// TIA Portal V21 export
FUNCTION "PHT_Logic" : Void   // FC1206, LAD
{ S7_Optimized_Access := 'FALSE' }
// stored: AutoNumber false, SetENOAutomatically false
   VAR_TEMP   // added for the SCL form of the ladder/FBD networks
      _w1 : Bool;
      _w2 : Bool;
      _w3 : Bool;
      _w4 : Bool;
      _w5 : Bool;
      _w6 : Bool;
      _w7 : Bool;
   END_VAR
BEGIN

REGION Network 1: "PHT Cycle".Start
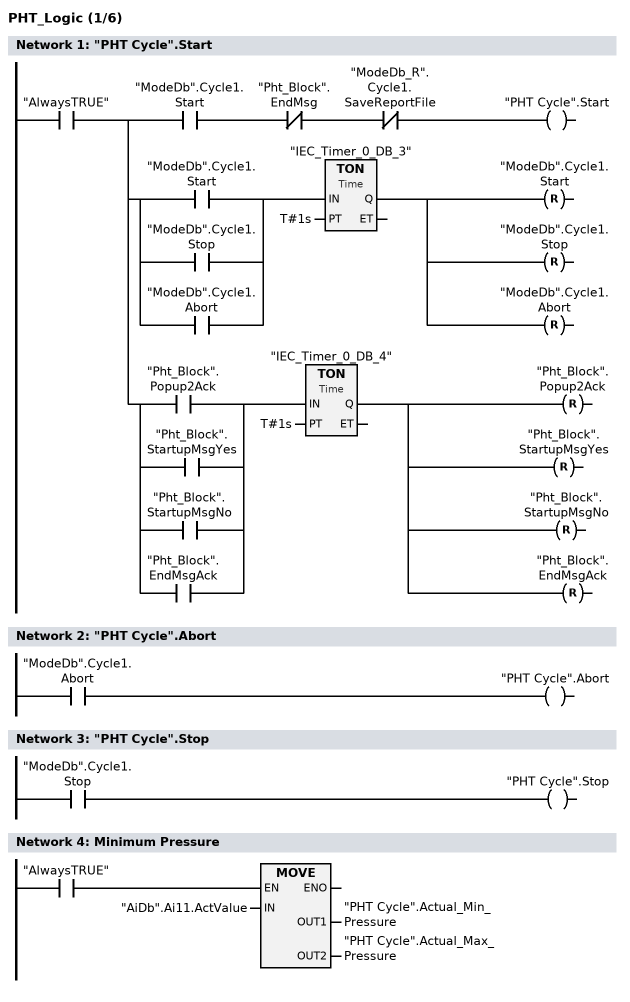
   RUNG wire#powerrail
      Contact( "AlwaysTRUE" )
      wire#w1
      Contact( "ModeDb".Cycle1.Start )
      I_Contact( "Pht_Block".EndMsg )
      I_Contact( "ModeDb_R".Cycle1.SaveReportFile )
      Coil( "PHT Cycle".Start )
   END_RUNG
   RUNG wire#w1
      Contact( "ModeDb".Cycle1.Start )
      wire#w2
      { S7_Templates := "time_type := Time" } "IEC_Timer_0_DB_3".TON(pt := T#1s, et =>)
      wire#w3
      R_Coil( "ModeDb".Cycle1.Start )
   END_RUNG
   RUNG wire#w1
      Contact( "ModeDb".Cycle1.Stop )
   END_RUNG wire#w2
   RUNG wire#w1
      Contact( "ModeDb".Cycle1.Abort )
   END_RUNG wire#w2
   RUNG wire#w3
      R_Coil( "ModeDb".Cycle1.Stop )
   END_RUNG
   RUNG wire#w3
      R_Coil( "ModeDb".Cycle1.Abort )
   END_RUNG
   RUNG wire#w1
      Contact( "Pht_Block".Popup2Ack )
      wire#w4
      { S7_Templates := "time_type := Time" } "IEC_Timer_0_DB_4".TON(pt := T#1s, et =>)
      wire#w5
      R_Coil( "Pht_Block".Popup2Ack )
   END_RUNG
   RUNG wire#w1
      Contact( "Pht_Block".StartupMsgYes )
   END_RUNG wire#w4
   RUNG wire#w1
      Contact( "Pht_Block".StartupMsgNo )
   END_RUNG wire#w4
   RUNG wire#w1
      Contact( "Pht_Block".EndMsgAck )
   END_RUNG wire#w4
   RUNG wire#w5
      R_Coil( "Pht_Block".StartupMsgYes )
   END_RUNG
   RUNG wire#w5
      R_Coil( "Pht_Block".StartupMsgNo )
   END_RUNG
   RUNG wire#w5
      R_Coil( "Pht_Block".EndMsgAck )
   END_RUNG
   // the same network as SCL:
   "PHT Cycle".Start := "AlwaysTRUE" AND "ModeDb".Cycle1.Start AND NOT "Pht_Block".EndMsg AND NOT "ModeDb_R".Cycle1.SaveReportFile;
   "IEC_Timer_0_DB_3".TON(IN := "AlwaysTRUE" AND ("ModeDb".Cycle1.Start OR "ModeDb".Cycle1.Stop OR "ModeDb".Cycle1.Abort),
                          PT := T#1s);
   IF "IEC_Timer_0_DB_3".Q THEN
       "ModeDb".Cycle1.Start := FALSE;
       "ModeDb".Cycle1.Stop := FALSE;
       "ModeDb".Cycle1.Abort := FALSE;
   END_IF;
   "IEC_Timer_0_DB_4".TON(IN := "AlwaysTRUE" AND ("Pht_Block".Popup2Ack OR "Pht_Block".StartupMsgYes OR "Pht_Block".StartupMsgNo OR "Pht_Block".EndMsgAck),
                          PT := T#1s);
   IF "IEC_Timer_0_DB_4".Q THEN
       "Pht_Block".Popup2Ack := FALSE;
       "Pht_Block".StartupMsgYes := FALSE;
       "Pht_Block".StartupMsgNo := FALSE;
       "Pht_Block".EndMsgAck := FALSE;
   END_IF;
END_REGION

REGION Network 2: "PHT Cycle".Abort
   RUNG wire#powerrail
      Contact( "ModeDb".Cycle1.Abort )
      Coil( "PHT Cycle".Abort )
   END_RUNG
   // the same network as SCL:
   "PHT Cycle".Abort := "ModeDb".Cycle1.Abort;
END_REGION

REGION Network 3: "PHT Cycle".Stop
   RUNG wire#powerrail
      Contact( "ModeDb".Cycle1.Stop )
      Coil( "PHT Cycle".Stop )
   END_RUNG
   // the same network as SCL:
   "PHT Cycle".Stop := "ModeDb".Cycle1.Stop;
END_REGION

REGION Network 4: Minimum Pressure
   RUNG wire#powerrail
      Contact( "AlwaysTRUE" )
      Move(in := "AiDb".Ai11.ActValue, out1 => "PHT Cycle".Actual_Min_Pressure, out2 => "PHT Cycle".Actual_Max_Pressure)
   END_RUNG
   // the same network as SCL:
   IF "AlwaysTRUE" THEN
       "PHT Cycle".Actual_Min_Pressure := "AiDb".Ai11.ActValue;
       "PHT Cycle".Actual_Max_Pressure := "AiDb".Ai11.ActValue;
   END_IF;
END_REGION

REGION Network 5: "PHT Cycle".fault
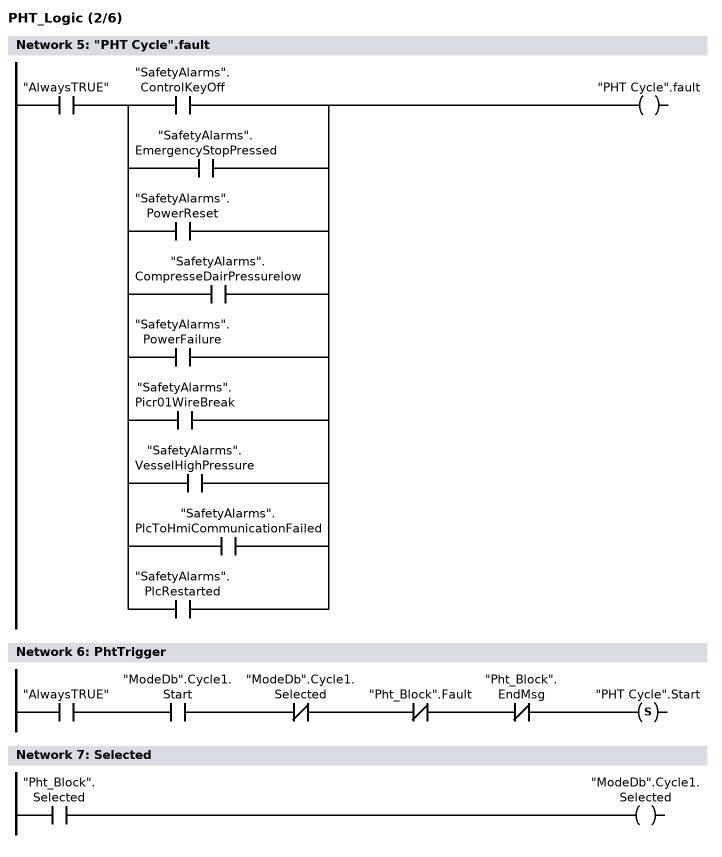
   RUNG wire#powerrail
      Contact( "AlwaysTRUE" )
      wire#w1
      Contact( "SafetyAlarms".ControlKeyOff )
      wire#w2
      Coil( "PHT Cycle".fault )
   END_RUNG
   RUNG wire#w1
      Contact( "SafetyAlarms".EmergencyStopPressed )
   END_RUNG wire#w2
   RUNG wire#w1
      Contact( "SafetyAlarms".PowerReset )
   END_RUNG wire#w2
   RUNG wire#w1
      Contact( "SafetyAlarms".CompresseDairPressurelow )
   END_RUNG wire#w2
   RUNG wire#w1
      Contact( "SafetyAlarms".PowerFailure )
   END_RUNG wire#w2
   RUNG wire#w1
      Contact( "SafetyAlarms".Picr01WireBreak )
   END_RUNG wire#w2
   RUNG wire#w1
      Contact( "SafetyAlarms".VesselHighPressure )
   END_RUNG wire#w2
   RUNG wire#w1
      Contact( "SafetyAlarms".PlcToHmiCommunicationFailed )
   END_RUNG wire#w2
   RUNG wire#w1
      Contact( "SafetyAlarms".PlcRestarted )
   END_RUNG wire#w2
   // the same network as SCL:
   "PHT Cycle".fault := "AlwaysTRUE" AND ("SafetyAlarms".ControlKeyOff OR "SafetyAlarms".EmergencyStopPressed OR "SafetyAlarms".PowerReset OR "SafetyAlarms".CompresseDairPressurelow OR "SafetyAlarms".PowerFailure OR "SafetyAlarms".Picr01WireBreak OR "SafetyAlarms".VesselHighPressure OR "SafetyAlarms".PlcToHmiCommunicationFailed OR "SafetyAlarms".PlcRestarted);
END_REGION

REGION Network 6: PhtTrigger
   RUNG wire#powerrail
      Contact( "AlwaysTRUE" )
      Contact( "ModeDb".Cycle1.Start )
      I_Contact( "ModeDb".Cycle1.Selected )
      I_Contact( "Pht_Block".Fault )
      I_Contact( "Pht_Block".EndMsg )
      S_Coil( "PHT Cycle".Start )
   END_RUNG
   // the same network as SCL:
   IF "AlwaysTRUE" AND "ModeDb".Cycle1.Start AND NOT "ModeDb".Cycle1.Selected AND NOT "Pht_Block".Fault AND NOT "Pht_Block".EndMsg THEN
       "PHT Cycle".Start := TRUE;
   END_IF;
END_REGION

REGION Network 7: Selected
   RUNG wire#powerrail
      Contact( "Pht_Block".Selected )
      Coil( "ModeDb".Cycle1.Selected )
   END_RUNG
   // the same network as SCL:
   "ModeDb".Cycle1.Selected := "Pht_Block".Selected;
END_REGION

REGION Network 8: PHT Block
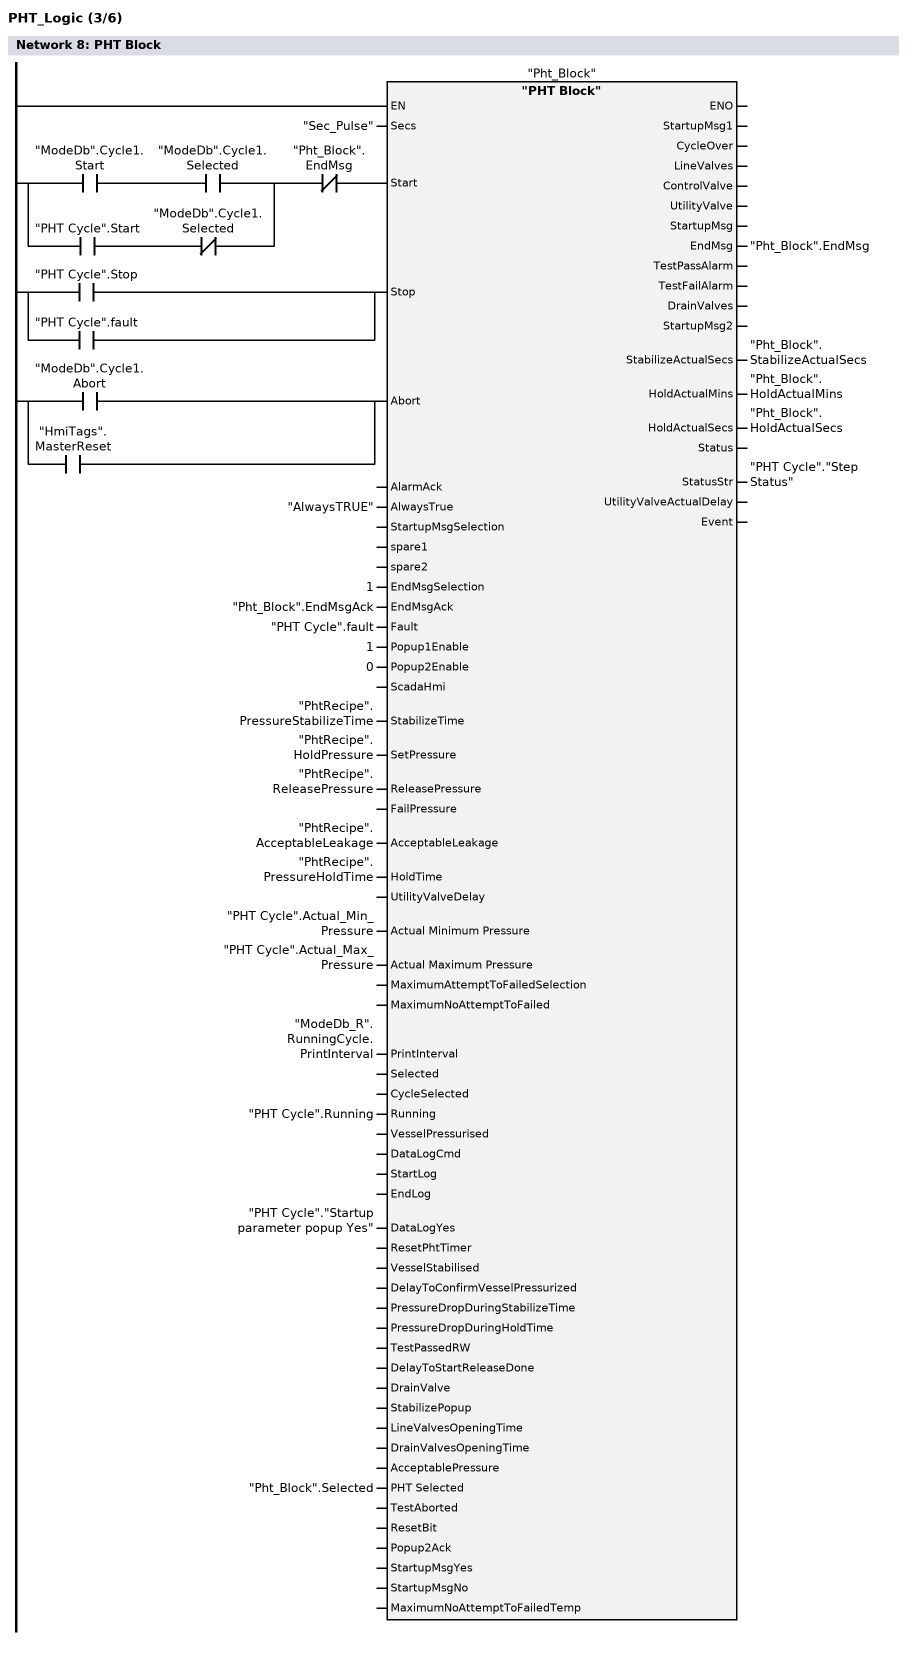
   RUNG wire#powerrail
      "Pht_Block"(Start := wire#w2, Stop := wire#w3, Abort := wire#w4, Secs := "Sec_Pulse", AlarmAck :=, AlwaysTrue := "AlwaysTRUE", StartupMsgSelection :=, spare1 :=, spare2 :=, EndMsgSelection := 1, EndMsgAck := "Pht_Block".EndMsgAck, Fault := "PHT Cycle".fault, Popup1Enable := 1, Popup2Enable := 0, ScadaHmi :=, StabilizeTime := "PhtRecipe".PressureStabilizeTime, SetPressure := "PhtRecipe".HoldPressure, ReleasePressure := "PhtRecipe".ReleasePressure, FailPressure :=, AcceptableLeakage := "PhtRecipe".AcceptableLeakage, HoldTime := "PhtRecipe".PressureHoldTime, UtilityValveDelay :=, "Actual Minimum Pressure" := "PHT Cycle".Actual_Min_Pressure, "Actual Maximum Pressure" := "PHT Cycle".Actual_Max_Pressure, MaximumAttemptToFailedSelection :=, MaximumNoAttemptToFailed :=, PrintInterval := "ModeDb_R".RunningCycle.PrintInterval, Selected :=, CycleSelected :=, Running := "PHT Cycle".Running, VesselPressurised :=, DataLogCmd :=, StartLog :=, EndLog :=, DataLogYes := "PHT Cycle"."Startup parameter popup Yes", ResetPhtTimer :=, VesselStabilised :=, DelayToConfirmVesselPressurized :=, PressureDropDuringStabilizeTime :=, PressureDropDuringHoldTime :=, TestPassedRW :=, DelayToStartReleaseDone :=, DrainValve :=, StabilizePopup :=, LineValvesOpeningTime :=, DrainValvesOpeningTime :=, AcceptablePressure :=, "PHT Selected" := "Pht_Block".Selected, TestAborted :=, ResetBit :=, Popup2Ack :=, StartupMsgYes :=, StartupMsgNo :=, MaximumNoAttemptToFailedTemp :=, StartupMsg1 =>, CycleOver =>, LineValves =>, ControlValve =>, UtilityValve =>, StartupMsg =>, EndMsg => "Pht_Block".EndMsg, TestPassAlarm =>, TestFailAlarm =>, DrainValves =>, StartupMsg2 =>, StabilizeActualSecs => "Pht_Block".StabilizeActualSecs, HoldActualMins => "Pht_Block".HoldActualMins, HoldActualSecs => "Pht_Block".HoldActualSecs, Status =>, StatusStr => "PHT Cycle"."Step Status", UtilityValveActualDelay =>, Event =>)
   END_RUNG
   RUNG wire#powerrail
      Contact( "ModeDb".Cycle1.Start )
      Contact( "ModeDb".Cycle1.Selected )
      wire#w1
      I_Contact( "Pht_Block".EndMsg )
   END_RUNG wire#w2
   RUNG wire#powerrail
      Contact( "PHT Cycle".Start )
      I_Contact( "ModeDb".Cycle1.Selected )
   END_RUNG wire#w1
   RUNG wire#powerrail
      Contact( "PHT Cycle".Stop )
   END_RUNG wire#w3
   RUNG wire#powerrail
      Contact( "PHT Cycle".fault )
   END_RUNG wire#w3
   RUNG wire#powerrail
      Contact( "ModeDb".Cycle1.Abort )
   END_RUNG wire#w4
   RUNG wire#powerrail
      Contact( "HmiTags".MasterReset )
   END_RUNG wire#w4
   // the same network as SCL:
   "Pht_Block"(Secs := "Sec_Pulse",   // "PHT Block"
               Start := (("ModeDb".Cycle1.Start AND "ModeDb".Cycle1.Selected) OR ("PHT Cycle".Start AND NOT "ModeDb".Cycle1.Selected)) AND NOT "Pht_Block".EndMsg,
               Stop := "PHT Cycle".Stop OR "PHT Cycle".fault,
               Abort := "ModeDb".Cycle1.Abort OR "HmiTags".MasterReset,
               AlwaysTrue := "AlwaysTRUE",
               EndMsgSelection := 1,
               EndMsgAck := "Pht_Block".EndMsgAck,
               Fault := "PHT Cycle".fault,
               Popup1Enable := 1,
               Popup2Enable := 0,
               StabilizeTime := "PhtRecipe".PressureStabilizeTime,
               SetPressure := "PhtRecipe".HoldPressure,
               ReleasePressure := "PhtRecipe".ReleasePressure,
               AcceptableLeakage := "PhtRecipe".AcceptableLeakage,
               HoldTime := "PhtRecipe".PressureHoldTime,
               "Actual Minimum Pressure" := "PHT Cycle".Actual_Min_Pressure,
               "Actual Maximum Pressure" := "PHT Cycle".Actual_Max_Pressure,
               PrintInterval := "ModeDb_R".RunningCycle.PrintInterval,
               Running := "PHT Cycle".Running,
               DataLogYes := "PHT Cycle"."Startup parameter popup Yes",
               "PHT Selected" := "Pht_Block".Selected,
               EndMsg => "Pht_Block".EndMsg,
               StabilizeActualSecs => "Pht_Block".StabilizeActualSecs,
               HoldActualMins => "Pht_Block".HoldActualMins,
               HoldActualSecs => "Pht_Block".HoldActualSecs,
               StatusStr => "PHT Cycle"."Step Status");
END_REGION

REGION Network 9: PHT ALARMS
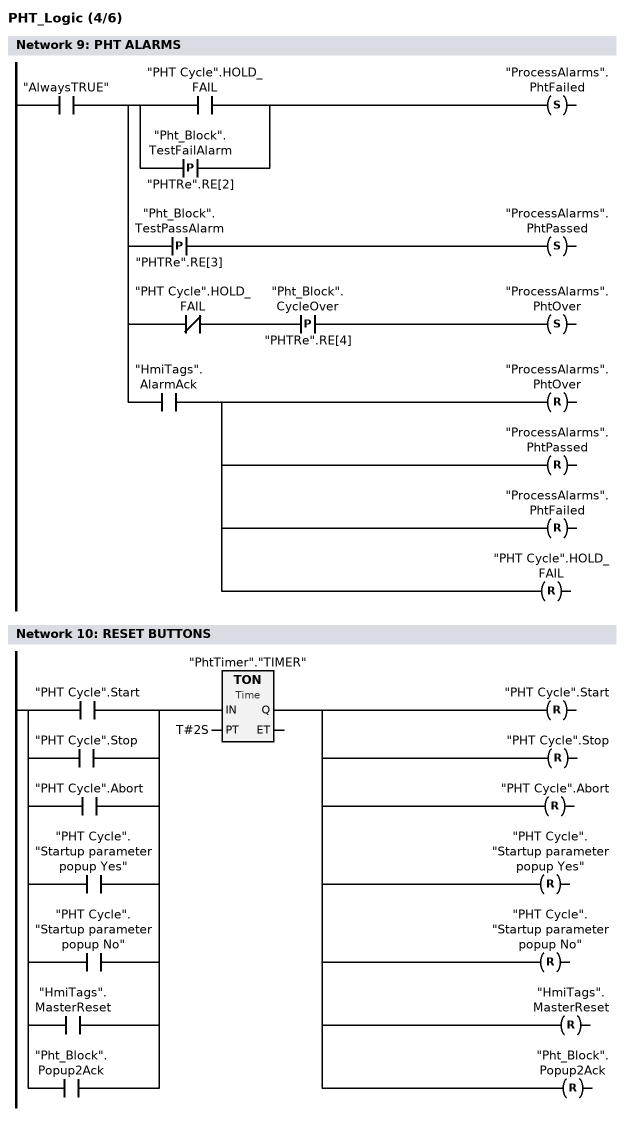
   RUNG wire#powerrail
      Contact( "AlwaysTRUE" )
      wire#w1
      Contact( "PHT Cycle".HOLD_FAIL )
      wire#w2
      S_Coil( "ProcessAlarms".PhtFailed )
   END_RUNG
   RUNG wire#w1
      P_Contact(operand := "Pht_Block".TestFailAlarm, bit := "PHTRe".RE[2])
   END_RUNG wire#w2
   RUNG wire#w1
      P_Contact(operand := "Pht_Block".TestPassAlarm, bit := "PHTRe".RE[3])
      S_Coil( "ProcessAlarms".PhtPassed )
   END_RUNG
   RUNG wire#w1
      I_Contact( "PHT Cycle".HOLD_FAIL )
      P_Contact(operand := "Pht_Block".CycleOver, bit := "PHTRe".RE[4])
      S_Coil( "ProcessAlarms".PhtOver )
   END_RUNG
   RUNG wire#w1
      Contact( "HmiTags".AlarmAck )
      wire#w3
      R_Coil( "ProcessAlarms".PhtOver )
   END_RUNG
   RUNG wire#w3
      R_Coil( "ProcessAlarms".PhtPassed )
   END_RUNG
   RUNG wire#w3
      R_Coil( "ProcessAlarms".PhtFailed )
   END_RUNG
   RUNG wire#w3
      R_Coil( "PHT Cycle".HOLD_FAIL )
   END_RUNG
   // the same network as SCL:
   #_w1 := "AlwaysTRUE" AND "Pht_Block".TestFailAlarm AND NOT "PHTRe".RE[2];   // rising edge of "Pht_Block".TestFailAlarm
   "PHTRe".RE[2] := "Pht_Block".TestFailAlarm;
   IF ("AlwaysTRUE" AND "PHT Cycle".HOLD_FAIL) OR #_w1 THEN "ProcessAlarms".PhtFailed := TRUE; END_IF;
   #_w2 := "AlwaysTRUE" AND "Pht_Block".TestPassAlarm AND NOT "PHTRe".RE[3];   // rising edge of "Pht_Block".TestPassAlarm
   "PHTRe".RE[3] := "Pht_Block".TestPassAlarm;
   IF #_w2 THEN "ProcessAlarms".PhtPassed := TRUE; END_IF;
   #_w3 := "AlwaysTRUE" AND NOT "PHT Cycle".HOLD_FAIL AND "Pht_Block".CycleOver AND NOT "PHTRe".RE[4];   // rising edge of "Pht_Block".CycleOver
   "PHTRe".RE[4] := "Pht_Block".CycleOver;
   IF #_w3 THEN "ProcessAlarms".PhtOver := TRUE; END_IF;
   IF "AlwaysTRUE" AND "HmiTags".AlarmAck THEN
       "ProcessAlarms".PhtOver := FALSE;
       "ProcessAlarms".PhtPassed := FALSE;
       "ProcessAlarms".PhtFailed := FALSE;
       "PHT Cycle".HOLD_FAIL := FALSE;
   END_IF;
END_REGION

REGION Network 10: RESET BUTTONS
   RUNG wire#powerrail
      Contact( "PHT Cycle".Start )
      wire#w1
      { S7_Templates := "time_type := Time" } "PhtTimer"."TIMER".TON(pt := T#2S, et =>)
      wire#w2
      R_Coil( "PHT Cycle".Start )
   END_RUNG
   RUNG wire#powerrail
      Contact( "PHT Cycle".Stop )
   END_RUNG wire#w1
   RUNG wire#powerrail
      Contact( "PHT Cycle".Abort )
   END_RUNG wire#w1
   RUNG wire#powerrail
      Contact( "PHT Cycle"."Startup parameter popup Yes" )
   END_RUNG wire#w1
   RUNG wire#powerrail
      Contact( "PHT Cycle"."Startup parameter popup No" )
   END_RUNG wire#w1
   RUNG wire#powerrail
      Contact( "HmiTags".MasterReset )
   END_RUNG wire#w1
   RUNG wire#powerrail
      Contact( "Pht_Block".Popup2Ack )
   END_RUNG wire#w1
   RUNG wire#w2
      R_Coil( "PHT Cycle".Stop )
   END_RUNG
   RUNG wire#w2
      R_Coil( "PHT Cycle".Abort )
   END_RUNG
   RUNG wire#w2
      R_Coil( "PHT Cycle"."Startup parameter popup Yes" )
   END_RUNG
   RUNG wire#w2
      R_Coil( "PHT Cycle"."Startup parameter popup No" )
   END_RUNG
   RUNG wire#w2
      R_Coil( "HmiTags".MasterReset )
   END_RUNG
   RUNG wire#w2
      R_Coil( "Pht_Block".Popup2Ack )
   END_RUNG
   // the same network as SCL:
   "PhtTimer"."TIMER".TON(IN := "PHT Cycle".Start OR "PHT Cycle".Stop OR "PHT Cycle".Abort OR "PHT Cycle"."Startup parameter popup Yes" OR "PHT Cycle"."Startup parameter popup No" OR "HmiTags".MasterReset OR "Pht_Block".Popup2Ack,
                          PT := T#2S);
   IF "PhtTimer"."TIMER".Q THEN
       "PHT Cycle".Start := FALSE;
       "PHT Cycle".Stop := FALSE;
       "PHT Cycle".Abort := FALSE;
       "PHT Cycle"."Startup parameter popup Yes" := FALSE;
       "PHT Cycle"."Startup parameter popup No" := FALSE;
       "HmiTags".MasterReset := FALSE;
       "Pht_Block".Popup2Ack := FALSE;
   END_IF;
END_REGION

REGION Network 11: RESULT
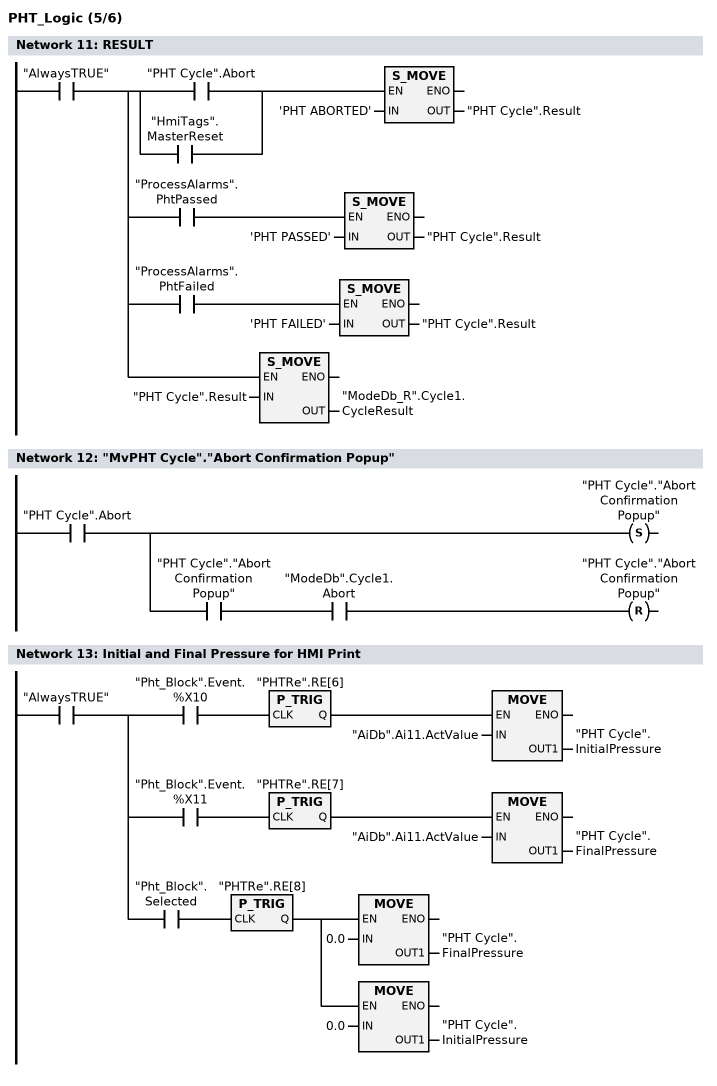
   RUNG wire#powerrail
      Contact( "AlwaysTRUE" )
      wire#w1
      Contact( "PHT Cycle".Abort )
      wire#w2
      S_Move(in := 'PHT ABORTED', out => "PHT Cycle".Result)
   END_RUNG
   RUNG wire#w1
      Contact( "HmiTags".MasterReset )
   END_RUNG wire#w2
   RUNG wire#w1
      Contact( "ProcessAlarms".PhtPassed )
      S_Move(in := 'PHT PASSED', out => "PHT Cycle".Result)
   END_RUNG
   RUNG wire#w1
      Contact( "ProcessAlarms".PhtFailed )
      S_Move(in := 'PHT FAILED', out => "PHT Cycle".Result)
   END_RUNG
   RUNG wire#w1
      S_Move(in := "PHT Cycle".Result, out => "ModeDb_R".Cycle1.CycleResult)
   END_RUNG
   // the same network as SCL:
   IF "AlwaysTRUE" AND ("PHT Cycle".Abort OR "HmiTags".MasterReset) THEN
       "PHT Cycle".Result := 'PHT ABORTED';
   END_IF;
   IF "AlwaysTRUE" AND "ProcessAlarms".PhtPassed THEN "PHT Cycle".Result := 'PHT PASSED'; END_IF;
   IF "AlwaysTRUE" AND "ProcessAlarms".PhtFailed THEN "PHT Cycle".Result := 'PHT FAILED'; END_IF;
   IF "AlwaysTRUE" THEN "ModeDb_R".Cycle1.CycleResult := "PHT Cycle".Result; END_IF;
END_REGION

REGION Network 12: "MvPHT Cycle"."Abort Confirmation Popup"
   RUNG wire#powerrail
      Contact( "PHT Cycle".Abort )
      wire#w1
      S_Coil( "PHT Cycle"."Abort Confirmation Popup" )
   END_RUNG
   RUNG wire#w1
      Contact( "PHT Cycle"."Abort Confirmation Popup" )
      Contact( "ModeDb".Cycle1.Abort )
      R_Coil( "PHT Cycle"."Abort Confirmation Popup" )
   END_RUNG
   // the same network as SCL:
   IF "PHT Cycle".Abort THEN "PHT Cycle"."Abort Confirmation Popup" := TRUE; END_IF;
   IF "PHT Cycle".Abort AND "PHT Cycle"."Abort Confirmation Popup" AND "ModeDb".Cycle1.Abort THEN
       "PHT Cycle"."Abort Confirmation Popup" := FALSE;
   END_IF;
END_REGION

REGION Network 13: Initial and Final Pressure for HMI Print
   RUNG wire#powerrail
      Contact( "AlwaysTRUE" )
      wire#w1
      Contact( "Pht_Block".Event.%X10 )
      P_Trig( "PHTRe".RE[6] )
      Move(in := "AiDb".Ai11.ActValue, out1 => "PHT Cycle".InitialPressure)
   END_RUNG
   RUNG wire#w1
      Contact( "Pht_Block".Event.%X11 )
      P_Trig( "PHTRe".RE[7] )
      Move(in := "AiDb".Ai11.ActValue, out1 => "PHT Cycle".FinalPressure)
   END_RUNG
   RUNG wire#w1
      Contact( "Pht_Block".Selected )
      P_Trig( "PHTRe".RE[8] )
      wire#w2
      Move(in := 0.0, out1 => "PHT Cycle".FinalPressure)
   END_RUNG
   RUNG wire#w2
      Move(in := 0.0, out1 => "PHT Cycle".InitialPressure)
   END_RUNG
   // the same network as SCL:
   #_w1 := "AlwaysTRUE" AND "Pht_Block".Event.%X10;
   #_w2 := #_w1 AND NOT "PHTRe".RE[6];   // rising edge
   "PHTRe".RE[6] := #_w1;
   IF #_w2 THEN "PHT Cycle".InitialPressure := "AiDb".Ai11.ActValue; END_IF;
   #_w3 := "AlwaysTRUE" AND "Pht_Block".Event.%X11;
   #_w4 := #_w3 AND NOT "PHTRe".RE[7];   // rising edge
   "PHTRe".RE[7] := #_w3;
   IF #_w4 THEN "PHT Cycle".FinalPressure := "AiDb".Ai11.ActValue; END_IF;
   #_w5 := "AlwaysTRUE" AND "Pht_Block".Selected;
   #_w6 := #_w5 AND NOT "PHTRe".RE[8];   // rising edge
   "PHTRe".RE[8] := #_w5;
   IF #_w6 THEN
       "PHT Cycle".FinalPressure := 0.0;
       "PHT Cycle".InitialPressure := 0.0;
   END_IF;
END_REGION

REGION Network 14: "PHT Cycle".HoldStartTimeLog
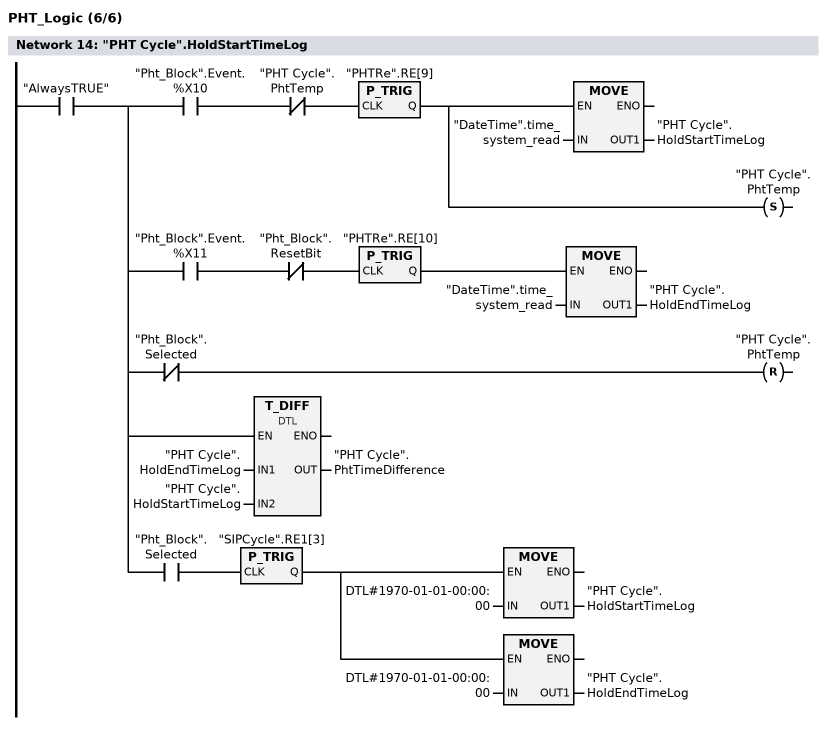
   RUNG wire#powerrail
      Contact( "AlwaysTRUE" )
      wire#w1
      Contact( "Pht_Block".Event.%X10 )
      I_Contact( "PHT Cycle".PhtTemp )
      P_Trig( "PHTRe".RE[9] )
      wire#w2
      Move(in := "DateTime".time_system_read, out1 => "PHT Cycle".HoldStartTimeLog)
   END_RUNG
   RUNG wire#w2
      S_Coil( "PHT Cycle".PhtTemp )
   END_RUNG
   RUNG wire#w1
      Contact( "Pht_Block".Event.%X11 )
      I_Contact( "Pht_Block".ResetBit )
      P_Trig( "PHTRe".RE[10] )
      Move(in := "DateTime".time_system_read, out1 => "PHT Cycle".HoldEndTimeLog)
   END_RUNG
   RUNG wire#w1
      I_Contact( "Pht_Block".Selected )
      R_Coil( "PHT Cycle".PhtTemp )
   END_RUNG
   RUNG wire#w1
      { S7_Templates := "[date_type := DTL, time_type := Time]" } T_DIFF(IN1 := "PHT Cycle".HoldEndTimeLog, IN2 := "PHT Cycle".HoldStartTimeLog, OUT => "PHT Cycle".PhtTimeDifference)
   END_RUNG
   RUNG wire#w1
      Contact( "Pht_Block".Selected )
      P_Trig( "SIPCycle".RE1[3] )
      wire#w3
      Move(in := DTL#1970-01-01-00:00:00, out1 => "PHT Cycle".HoldStartTimeLog)
   END_RUNG
   RUNG wire#w3
      Move(in := DTL#1970-01-01-00:00:00, out1 => "PHT Cycle".HoldEndTimeLog)
   END_RUNG
   // the same network as SCL:
   #_w1 := "AlwaysTRUE" AND "Pht_Block".Event.%X10 AND NOT "PHT Cycle".PhtTemp;
   #_w2 := #_w1 AND NOT "PHTRe".RE[9];   // rising edge
   "PHTRe".RE[9] := #_w1;
   IF #_w2 THEN
       "PHT Cycle".HoldStartTimeLog := "DateTime".time_system_read;
       "PHT Cycle".PhtTemp := TRUE;
   END_IF;
   #_w3 := "AlwaysTRUE" AND "Pht_Block".Event.%X11 AND NOT "Pht_Block".ResetBit;
   #_w4 := #_w3 AND NOT "PHTRe".RE[10];   // rising edge
   "PHTRe".RE[10] := #_w3;
   IF #_w4 THEN "PHT Cycle".HoldEndTimeLog := "DateTime".time_system_read; END_IF;
   IF "AlwaysTRUE" AND NOT "Pht_Block".Selected THEN "PHT Cycle".PhtTemp := FALSE; END_IF;
   #_w5 := "AlwaysTRUE";
   IF #_w5 THEN
       T_DIFF(IN1 := "PHT Cycle".HoldEndTimeLog,
              IN2 := "PHT Cycle".HoldStartTimeLog,
              OUT => "PHT Cycle".PhtTimeDifference);
   END_IF;
   #_w6 := #_w5 AND "Pht_Block".Selected;
   #_w7 := #_w6 AND NOT "SIPCycle".RE1[3];   // rising edge
   "SIPCycle".RE1[3] := #_w6;
   IF #_w7 THEN
       "PHT Cycle".HoldStartTimeLog := DTL#1970-01-01-00:00:00;
       "PHT Cycle".HoldEndTimeLog := DTL#1970-01-01-00:00:00;
   END_IF;
END_REGION

REGION Network 15 (SCL): SCL ROUNDOFF
   // Step 1: get TIME
   "PHT Cycle".TempTime := "PHT Cycle".PhtTimeDifference;

   // Step 2: TIME → milliseconds
   "PHT Cycle".TempMs := TIME_TO_DINT("PHT Cycle".TempTime);

   // Step 3: make positive (optional)
   //"PHT Cycle".TempMs := ABS("PHT Cycle".TempMs);

   // Step 4: ROUND milliseconds to seconds
   "PHT Cycle".TotalSecondsTag := ("PHT Cycle".TempMs + 500) / 1000;

   // Step 5: split HH MM SS
   "PHT Cycle".Hours := DINT_TO_INT("PHT Cycle".TotalSecondsTag / 3600);

   "PHT Cycle".Minutes := DINT_TO_INT(
   ("PHT Cycle".TotalSecondsTag MOD 3600) / 60
   );

   "PHT Cycle".Seconds := DINT_TO_INT(
    "PHT Cycle".TotalSecondsTag MOD 60
   );
END_REGION
END_FUNCTION
